// TIA Portal V20 export
TYPE "UDT_MTP_ProcedureHealthView"
   STRUCT
      WQC { ExternalWritable := 'False'} : Byte := 16#FF;   // Worst Quality Code
      CommandInfo { ExternalWritable := 'False'} : DWord := 16#FFFFFFFF;   // command info variable
   END_STRUCT;
END_TYPE
